# EPICS autosave request: iocBoot/iocagilent33521a/auto_settings_agilent33521a.req
file "agilent33521a_settings.req",                P=$(P),  R=$(R)
